### Bounded Queue Example (overwriteEnabled = FALSE)
```iecst
// Buffer capacity = 3
value := 100; ring.Push(value);  // Buffer: [100], returns TRUE
value := 200; ring.Push(value);  // Buffer: [100, 200], returns TRUE
value := 300; ring.Push(value);  // Buffer: [100, 200, 300], returns TRUE

// Push to full buffer fails
value := 400;
success := ring.Push(value);     // Returns FALSE, logs error, buffer unchanged
```

### Return Value
- **TRUE**: Element was successfully pushed to the ring buffer
- **FALSE**: Push operation failed (see error conditions)

### Error Conditions (both modes)
- Returns FALSE and logs error if buffer was not initialized
- Returns FALSE and logs error if element size doesn't match buffer element size
- Returns FALSE and logs error if underlying WriteAtIndex operation fails

### Error Conditions (overwriteEnabled = FALSE only)
- Returns FALSE and logs error if ring buffer is full (no available capacity)

### Parameters
- **element**: Must be a writable variable (not a literal) of the correct size
  - Must match the buffer's configured element size
  - Value will be copied into the ring buffer

### Side Effects (when not full)
- Adds one element to the ring buffer using WriteAtIndex
- Increments elementCount by 1 (managed by RingBuffer, not AnyBuffer)
- Advances tail pointer circularly
- Logs verbose trace message on success
- Logs error trace message on failure

### Side Effects (when full and overwriteEnabled = TRUE)
- Overwrites element at tail position using WriteAtIndex (no shifting!)
- Advances both head pointer and tail pointer circularly
- Element count remains at maximum capacity
- No physical element movement occurs
- No AnyBuffer counter modifications
- Logs verbose trace message on success

### Performance Considerations
- **When not full**: O(1) - uses WriteAtIndex (raw write, no counter overhead)
- **When full**: O(1) - uses WriteAtIndex with circular indexing (no shifting!)
- **Overall**: True O(1) constant-time operation for all scenarios
- **Optimal efficiency**: WriteAtIndex bypasses AnyBuffer counter management
- Ideal for high-frequency streaming and real-time data processing
*)
Push := FALSE;
IF NOT isInitialized THEN
	Trace.Error(__POUNAME(), 'Buffer was not initialized yet, execute method .init() at least once');
	RETURN;
END_IF

// valid sized element pushed?
IF element.diSize <> anyBuffer.Configuration.elementSize THEN
	Trace.Error(__POUNAME(), 'Pushed element is of improper size');
	RETURN;
END_IF

// Handle push based on buffer state
IF anyBuffer.Metadata.elementCount < anyBuffer.Configuration.capacity THEN
	// Buffer not yet full - use WriteAtIndex for direct write without counter changes
	Push := anyBuffer.ReplaceAtIndex(anyBuffer.Metadata.tailIndex, element);
	IF Push THEN
		// Advance tail circular
		AdvanceTail();

		// Replace index does not change counters, do it manually
		anyBuffer.Metadata.elementCount := anyBuffer.Metadata.elementCount + 1;
		anyBuffer.Metadata.capacity		:= anyBuffer.Metadata.capacity - 1;
	END_IF
ELSIF _overwrite THEN
	// Buffer is full and overwrite enabled - use WriteAtIndex for circular overwrite (no shifting!)
	Push := anyBuffer.ReplaceAtIndex(anyBuffer.Metadata.tailIndex, element);
	IF Push THEN
		// Advance tail circular
		AdvanceTail();

		// Advance head circular
		AdvanceHead();

		// elementCount stays at capacity
	END_IF
ELSE
	// Overwrite disabled - reject push when full (bounded queue behavior)
	Trace.Error(__POUNAME(), 'Attempt to push to full buffer with overwrite disabled');
	RETURN;
END_IF

// Push was ok, trace message
IF Push THEN
	Trace.Verbose(__POUNAME(), 'executed');
ELSE
	Trace.Error(__POUNAME(), 'FAILED');
END_IF
END_METHOD

END_FUNCTION_BLOCK

// Utilities/File/Interface/I_FileHandler
INTERFACE I_FileHandler EXTENDS I_Component, I_Cyclic, I_TaskResult, I_TaskResult, I_Resettable

METHOD ClearDocument
VAR_INPUT
END_VAR
END_METHOD

PROPERTY Datatype : T_MaxString
SET
END_SET
END_PROPERTY

METHOD LoadFile
END_METHOD

PROPERTY nData : UDINT
SET
END_SET
END_PROPERTY

PROPERTY PUBLIC Path : T_MaxString
GET
END_GET
SET
END_SET
END_PROPERTY

PROPERTY pData : PVOID
SET
END_SET
END_PROPERTY

METHOD ReadSymbol
END_METHOD

METHOD SaveFile
END_METHOD

PROPERTY SymbolName : T_MaxString
SET
END_SET
END_PROPERTY

PROPERTY Timeout : TIME
SET
END_SET
END_PROPERTY

METHOD UpdateSymbol
END_METHOD

END_INTERFACE

// Utilities/File/File_HMI
FUNCTION_BLOCK File_HMI EXTENDS HmiFunction
VAR
	File : I_FileHandler;
	{ attribute 'TcHmiSymbol.AddSymbol' }
	{ attribute 'TcHmiSymbol.AddSymbol.UserGroups' := '__SystemAdministrators,Admin' }
	File_HMI : ST_File_HMI;
END_VAR

PROPERTY LoadPermissive : I_Permissive
GET
LoadPermissive := File_HMI.Load.Permissive;
END_GET
END_PROPERTY

PROPERTY SavePermissive : I_Permissive
GET
SavePermissive := File_HMI.Save.Permissive;
END_GET
END_PROPERTY

PROPERTY ControlObject : I_Base
SET
__QueryInterface(ControlObject,File);
END_SET
END_PROPERTY

METHOD CyclicLogic
VAR_INST
	SaveRT		 : R_TRIG;
	LoadRT		 : R_TRIG;
	ReloadActive : BOOL;
END_VAR
IF File = 0 THEN
	RETURN;
END_IF

File_HMI.Name		:= File.Name;
File_HMI.HmiEnabled := Enabled;
// HMI Commands
IF Enabled THEN
	SaveRT(CLK := File_HMI.Save.Active);
	IF SaveRT.Q THEN
		IF File_HMI.Save.Permissive.OK THEN
			File.UpdateSymbol();
		END_IF
	END_IF

	IF ReloadActive AND NOT File.Busy AND NOT File.Error THEN
		File.ReadSymbol();
		ReloadActive := FALSE;
	END_IF

	LoadRT(CLK := File_HMI.Load.Active);
	IF LoadRT.Q THEN
		IF File_HMI.Load.Permissive.OK THEN
			File.LoadFile();
			ReloadActive := TRUE;
		END_IF
	END_IF

	IF File_HMI.NewPath THEN
		File.Path		 := File_HMI.Path;
		File_HMI.NewPath := FALSE;
	END_IF
END_IF
END_METHOD

(*FB_Init is always available implicitly and it is used primarily for initialization.
The return value is not evaluated. For a specific influence, you can also declare the
methods explicitly and provide additional code there with the standard initialization
code. You can evaluate the return value.*)
METHOD FB_Init : BOOL
VAR_INPUT
	(* TRUE: the retain variables are initialized (reset warm / reset cold)*)
	bInitRetains : BOOL;

	(* TRUE: the instance will be copied to the copy code afterward (online change)   *)
	bInCopyCode : BOOL;
	Name		: Core.T_MaxString;
	File		: I_FileHandler;
END_VAR
THIS^.File	:= File;
ControlType := 'File';
LinkObject	:= 'File_HMI';
END_METHOD

END_FUNCTION_BLOCK

// Utilities/File/JsonFile
FUNCTION_BLOCK JsonFile
VAR_GENERIC CONSTANT
	FileSize : UDINT := 10000;
END_VAR
EXTENDS CyclicComponent IMPLEMENTS I_FileHandler
VAR
	{attribute 'hide'}
	_Error : BOOL;
	{attribute 'hide'}
	_ErrorId : UDINT;

	//
	_Path	   : STRING;
	TonTimeout : TON;
	_Timeout   : TIME := T#1S;
	SeqLoad	   : UDINT;
	SeqSave	   : UDINT;

	// Folder Management
	CreateDir	 : FB_CreateDir;
	StringHelper : StringHelper;

	// Symbol
	JsonReadWriteDataType : FB_JsonReadWriteDatatype;
	ValueJson			  : STRING(FileSize);
	hr					  : HRESULT;
	_Datatype			  : T_MaxString;
	_SymbolName			  : T_MaxString;
	_nData				  : UDINT;
	_pData				  : PVOID;

	// Json Management 
	FileRead			  : BOOL;
	FileSave			  : BOOL;
	FileLoadOK			  : BOOL;
	FileSaveOK			  : BOOL;
	JsonFileMachineConfig : FB_JsonDomParser;
	JsonDoc				  : SJsonValue;
	JsonProp			  : SJsonValue;
END_VAR

METHOD CyclicLogic
IF _Path <> '' THEN
	FileLoadOK := JsonFileMachineConfig.LoadDocumentFromFile(sFile := _Path, bExec := FileRead);
	FileSaveOK := JsonFileMachineConfig.SaveDocumentToFile(sFile := _Path, bExec := FileSave);
END_IF

TonTimeout(IN := Busy, PT := _Timeout);
IF TonTimeout.Q THEN
	_Error := TRUE;
END_IF

SaveFileSequence();
LoadFileSequence();
END_METHOD

METHOD ClearDocument
VAR_INPUT
END_VAR
JsonDoc := JsonFileMachineConfig.NewDocument();
END_METHOD

PROPERTY Datatype : T_MaxString
SET
_Datatype := Datatype;
END_SET
END_PROPERTY

METHOD LoadFile
IF _Path = '' THEN
	_Error := TRUE;
	Trace.LogMessage(Name, 'File Path not set!');
	RETURN;
END_IF

IF Busy THEN
	RETURN;
END_IF

FileRead := TRUE;
SeqLoad	 := 10;
END_METHOD

PROPERTY nData : UDINT
SET
_nData := nData;
END_SET
END_PROPERTY

PROPERTY PUBLIC Path : T_MaxString
GET
Path := _Path;
END_GET
SET
//Prevent the path from have a space at the end
_Path := Path;
WHILE RIGHT(_Path, 1) = ' ' DO
	_Path := DELETE(_Path, 1, LEN(_Path));
END_WHILE
END_SET
END_PROPERTY

PROPERTY pData : PVOID
SET
_pData := pData;
END_SET
END_PROPERTY

METHOD ReadSymbol
IF JsonDoc = 0 THEN
	Trace.LogMessage(Name, 'Document File not loaded!');
	RETURN;
END_IF

IF _Datatype = '' THEN
	Trace.LogMessage(Name, 'No Datatype specified!');
	RETURN;
END_IF

IF _nData = 0 THEN
	Trace.LogMessage(Name, 'No nData specified!');
	RETURN;
END_IF

IF _pData = 0 THEN
	Trace.LogMessage(Name, 'No pData specified!');
	RETURN;
END_IF

IF _SymbolName = '' THEN
	Trace.LogMessage(Name, 'No PropertyName specified!');
	RETURN;
END_IF

IF Busy THEN
	RETURN;
END_IF

JsonProp := JsonFileMachineConfig.FindMemberPath(JsonDoc, _SymbolName);
JsonFileMachineConfig.CopyJson(v := JsonProp, pDoc := ValueJson, nDoc := SIZEOF(ValueJson));
IF JsonProp <> 0 THEN
	JsonReadWriteDataType.SetSymbolFromJson(sJson		:= ValueJson,
											sDataType	:= _Datatype,
											nData		:= _nData,
											pData		:= _pData,
											hrErrorCode => hr);
ELSE
	THIS^.UpdateSymbol();
END_IF
END_METHOD

METHOD SaveFile
IF _Path = '' THEN
	_Error := TRUE;
	Trace.LogMessage(Name, 'File Path not set!');
	RETURN;
END_IF

IF Busy THEN
	RETURN;
END_IF

FileSave := TRUE;
SeqSave	 := 10;
END_METHOD

PROPERTY SymbolName : T_MaxString
SET
_SymbolName := SymbolName;
END_SET
END_PROPERTY

PROPERTY Timeout : TIME
SET
_Timeout := Timeout;
END_SET
END_PROPERTY

METHOD UpdateSymbol
IF JsonDoc = 0 THEN
	Trace.LogMessage(Name, 'Document File not loaded!');
	RETURN;
END_IF

IF _Datatype = '' THEN
	Trace.LogMessage(Name, 'No Datatype specified!');
	RETURN;
END_IF

IF _nData = 0 THEN
	Trace.LogMessage(Name, 'No nData specified!');
	RETURN;
END_IF

IF _pData = 0 THEN
	Trace.LogMessage(Name, 'No pData specified!');
	RETURN;
END_IF

IF _SymbolName = '' THEN
	Trace.LogMessage(Name, 'No PropertyName specified!');
	RETURN;
END_IF

IF Busy THEN
	RETURN;
END_IF

// Create Json
JsonReadWriteDataType.CopyJsonStringFromSymbol(sDatatype   := _Datatype,
											   nData	   := _nData,
											   pData	   := _pData,
											   pDoc		   := ValueJson,
											   nDoc		   := SIZEOF(ValueJson),
											   hrErrorCode => hr);

// Attempt to find Member
jsonProp := JsonFileMachineConfig.FindMemberPath(JsonDoc, _SymbolName);
IF JsonProp <> 0 THEN
	JsonFileMachineConfig.SetJson(JsonProp, ValueJson);
ELSE
	JsonFileMachineConfig.AddJsonMember(JsonDoc, _SymbolName, ValueJson);
END_IF

// Save the update to file
FileSave := TRUE;
SeqSave	 := 10;
JsonProp := 0;
END_METHOD

METHOD PRIVATE LoadFileSequence
VAR_INST
	dirPath	 : T_MaxString;
	tryAgain : BOOL;
END_VAR

VAR
	msg : STRING;
END_VAR
CASE SeqLoad OF
	0:										// Attempt to Load File -> Command started in LoadFile()
	10:										// Load File Done
		IF NOT FileRead AND FileLoadOK THEN // File Found
			JsonDoc := JsonFileMachineConfig.GetDocumentRoot();
			SeqLoad := 0;
		END_IF

		IF (NOT FileRead AND NOT FileLoadOK) OR TonTimeout.Q THEN // File not Found
			tryAgain := FALSE;
			FileRead := FALSE;
			SeqLoad	 := 20;
		END_IF

	20:								  (*File Not Found - Create Directory if not exists*) ;
		CreateDir(bExecute := FALSE); //Prepare for rising edge in next step
		IF NOT tryAgain THEN
			dirPath := StringHelper.GetPath(_Path);
		ELSE
			dirPath := StringHelper.GetPath(dirPath);
		END_IF

		SeqLoad := 30;

	30:
		CreateDir(sNetId	:= '',
				  sPathName := dirPath,
				  ePath		:= PATH_GENERIC,
				  bExecute	:= TRUE);

		IF NOT CreateDir.bBusy THEN
			IF NOT CreateDir.bError THEN
				IF NOT tryAgain THEN
					SeqLoad := 40;
				ELSE
					tryAgain := FALSE;
					SeqLoad	 := 20;
				END_IF
			ELSE
				IF (CreateDir.nErrId = 1827) OR (CreateDir.nErrId = 1807) THEN
					//0x723 Folder is already existing or invalid sPathName or ePath parameter.
					msg := CONCAT(_Path, ' File not found, but folder is existing. File will be created');
					Trace.LogMessage(Name, msg);
					SeqLoad := 40;
				ELSIF CreateDir.nErrId = 1804 THEN
					//0x70C Folder not found.
					msg := CONCAT('Folder is not found: ', dirPath);
					msg := CONCAT(msg, ' Reducing Path and trying again.');
					Trace.LogMessage(Name, msg);
					tryagain := TRUE;

					// SeqLoad	 := 20; TwinCat Bug - Ticket BTS-168764 Germany
					SeqLoad := 40;
				ELSE
					msg := CONCAT('Create Directory Error: ', UDINT_TO_STRING(CreateDir.nErrId));
					Trace.LogMessage(Name, msg);
					SeqLoad := 999;
				END_IF
			END_IF
		END_IF

	40: // File not found -> Create file
		JsonDoc	 := JsonFileMachineConfig.NewDocument();
		FileSave := TRUE;
		SeqLoad	 := 50;

	50: // New Document Saved
		IF NOT FileSave AND FileSaveOk THEN
			_Error	:= FALSE;
			SeqLoad := 0;
		END_IF
END_CASE
END_METHOD

METHOD PRIVATE SaveFileSequence
CASE SeqSave OF
	0:	// Attempt to save File -> Command started in UpdateXYZ()
	10: // New Document Saved
		IF NOT FileSave AND FileSaveOk THEN
			SeqSave := 0;
		END_IF
END_CASE
END_METHOD

METHOD Reset
_Error		  := FALSE;
_ErrorId	  := 0;
SeqSave		  := 0;
SeqLoad		  := 0;
TonTimeout.IN := FALSE;
END_METHOD

{attribute 'monitoring' := 'call'}
PROPERTY Busy : BOOL
GET
Busy := SeqSave <> 0 OR SeqLoad <> 0;
END_GET
END_PROPERTY

{attribute 'monitoring' := 'call'}
PROPERTY Error : BOOL
GET
Error := _Error;
END_GET
END_PROPERTY

{attribute 'monitoring' := 'call'}
PROPERTY ErrorId : UDINT
GET
ErrorID := _ErrorID;
END_GET
END_PROPERTY

END_FUNCTION_BLOCK

// Utilities/File/StringHelper
{attribute 'no_explicit_call' := 'This FB is a CLASS and must be accessed using methods or properties'}
FUNCTION_BLOCK StringHelper

METHOD PROTECTED GetExtensionOrVarName : T_MaxString
VAR_INPUT
	input : T_MaxString;
END_VAR

VAR
	i		 : INT;
	charArry : ARRAY[0..255] OF STRING(1);
END_VAR
IF NOT ValidInput(input) THEN
	RETURN;
END_IF

charArry := StringToCharArray(input);
//Get Location of final delimiter '.'
FOR i := LEN(input) - 1 TO 0 BY -1 DO //Start at the end and find the last delimiter
	IF charArry[i] = '.' THEN
		GetExtensionOrVarName := RIGHT(input, LEN(input) - 1 - i);
		EXIT;
	END_IF
END_FOR
END_METHOD

METHOD PROTECTED GetFileNameFromPath : T_MaxString
VAR_INPUT
	input : T_MaxString;
END_VAR

VAR
	i			  : INT;
	searchResults : ARRAY[0..99] OF INT;
	tempPath	  : T_MaxString;
END_VAR
IF NOT ValidInput(input) THEN
	RETURN;
END_IF

tempPath := input; //Copy to temp variable for modification
FOR i := 0 TO LEN(input) - 1 DO
	searchResults[i] := FIND(tempPath, '\');
	IF searchResults[i] > 0 THEN
		tempPath := RIGHT(tempPath, LEN(tempPath) - searchResults[i]); //Remove begining up to and including the first delimiter
	ELSE
		EXIT; //No more delimiters remaining
	END_IF
END_FOR

GetFileNameFromPath := tempPath;
END_METHOD

METHOD PROTECTED GetFilePath : T_MaxString
VAR_INPUT
	input : T_MaxString;
END_VAR

VAR
	tempPath	  : T_MaxString;
	i			  : INT;
	searchResults : ARRAY[0..99] OF INT;
	location	  : INT;
END_VAR
IF NOT ValidInput(input) THEN
	RETURN;
END_IF

tempPath := input;								 //Copy to temp variable for modification
tempPath := LEFT(tempPath, (LEN(tempPath) - 1)); //Remove Last Character, on first pass this has no effect, but on subsequents passes this will remove the ending \

//Reduce String by removing each delimiter and counting number of characters removed to find last '\'
FOR i := 0 TO LEN(input) - 1 DO
	searchResults[i] := FIND(tempPath, '\');
	IF searchResults[i] > 0 THEN
		tempPath := RIGHT(tempPath, LEN(tempPath) - searchResults[i]); //Remove begining up to and including the first delimiter
	ELSE
		EXIT; //No more delimiters remaining
	END_IF
END_FOR

//Sum length of string to last delimiter
FOR i := 0 TO LEN(input) - 1 DO
	IF searchResults[i] > 0 THEN
		location := location + searchResults[i]; //Location of last delimiter
	ELSE
		EXIT;
	END_IF
END_FOR

GetFilePath := LEFT(input, location);
END_METHOD

METHOD GetName : T_MaxString
VAR_INPUT
	FullPath : T_MaxString;
END_VAR
IF NOT ValidInput(FullPath) THEN
	RETURN;
END_IF

//Find the First \ or . to determine if this is a File Path or Symbol Path
IF FIND(FullPath, '\') > 0 THEN
	GetName := GetFileNameFromPath(FullPath);
ELSE //symbolPath
	GetName := GetExtensionOrVarName(FullPath);
END_IF
END_METHOD

METHOD GetPath : T_MaxString
VAR_INPUT
	FullPath : T_MaxString;
END_VAR

VAR
	tempPath : T_MaxString;
END_VAR
IF NOT ValidInput(FullPath) THEN
	RETURN;
END_IF

//Find the First \ or . to determine if this is a File Path or Symbol Path
IF FIND(FullPath, '\') > 0 THEN
	GetPath := GetFilePath(FullPath);
ELSE //symbolPath
	GetPath := GetSymbolPath(FullPath);
END_IF
END_METHOD

METHOD PROTECTED GetSymbolPath : T_MaxString
VAR_INPUT
	input : T_MaxString;
END_VAR

VAR
	i		 : INT;
	charArry : ARRAY[0..255] OF STRING(1);
	tempPath : T_MaxString;
END_VAR
IF NOT ValidInput(input) THEN
	RETURN;
END_IF

charArry := StringToCharArray(input);
tempPath := input;					  //Copy to temp variable for modification
FOR i := LEN(input) - 1 TO 0 BY -1 DO //Start at the end and find the last delimiter
	IF charArry[i] = '.' THEN
		tempPath := LEFT(tempPath, i);
		EXIT;
	END_IF
END_FOR

GetSymbolPath := tempPath;
END_METHOD

METHOD PROTECTED RemoveFirstChar : T_MaxString
VAR_INPUT
	input : T_MaxString;
END_VAR
RemoveFirstChar := DELETE(input, 1, 1);
END_METHOD

METHOD PROTECTED RemoveLastChar : T_MaxString
VAR_INPUT
	input : T_MaxString;
END_VAR
RemoveLastChar := DELETE(input, 1, len(input));
END_METHOD

METHOD PROTECTED StringToCharArray : ARRAY[0..255] OF STRING(1)
VAR_INPUT
	input : T_MaxString;
END_VAR

VAR
	i		 : INT;
	end		 : INT;
	tempPath : T_MaxString;
END_VAR
IF NOT ValidInput(input) THEN
	RETURN;
END_IF

tempPath := input;
//Convert String to CharArray
FOR i := 0 TO LEN(input) - 1 DO
	StringToCharArray[i] := Left(tempPath, 1); //Return the first/next character
	tempPath			 := RemoveFirstChar(tempPath);
END_FOR
END_METHOD

METHOD PROTECTED ValidInput : BOOL
VAR_INPUT
	input : T_MaxString;
END_VAR
IF LEN(input) > 0 THEN
	ValidInput := TRUE;
ELSE
	ValidInput := FALSE;
END_IF
END_METHOD

END_FUNCTION_BLOCK

// Utilities/Flash/SyncedSquareWaves
FUNCTION_BLOCK SyncedSquareWaves EXTENDS CyclicComponent IMPLEMENTS I_Initializable
VAR
	_Initialized  : BOOL;
	PLC_CycleTime : UDINT;
	CycleTime_ms  : LREAL;

	//
	{attribute 'hide'}
	_Wave_500Hz : BOOL;
	{attribute 'hide'}
	_Wave_100Hz : BOOL;
	{attribute 'hide'}
	_Wave_50Hz : BOOL;
	{attribute 'hide'}
	_Wave_5Hz : BOOL;
	{attribute 'hide'}
	_Wave_2Hz : BOOL;
	{attribute 'hide'}
	_Wave_1Hz : BOOL;
	{attribute 'hide'}
	_Wave_0_5Hz : BOOL;
END_VAR

METHOD Initialize
//PLC Scan Info
PLC_CycleTime := TwinCAT_SystemInfoVarList._TaskInfo[GETCURTASKINDEXEX()].CycleTime;
CycleTime_ms  := TO_LREAL(PLC_CycleTime) / 10000.0;

//
_Wave_500Hz	 := TRUE;
_Wave_100Hz	 := TRUE;
_Wave_50Hz	 := TRUE;
_Wave_5Hz	 := TRUE;
_Wave_2Hz	 := TRUE;
_Wave_1Hz	 := TRUE;
_Wave_0_5Hz	 := TRUE;
_Initialized := TRUE;
END_METHOD

{attribute 'monitoring' := 'call'}
PROPERTY Initialized : BOOL
GET
Initialized := _Initialized;
END_GET
SET
_Initialized := Initialized;
END_SET
END_PROPERTY

//! @summary This method serves as the entry point for all underlying FB logic
METHOD PUBLIC CyclicLogic
VAR
	Counter		   : LREAL;
	CountsRequired : LREAL;
	CycleCount	   : UDINT;
END_VAR
IF NOT _Initialized THEN
	Initialize();
	RETURN;
END_IF

CycleCount := TwinCAT_SystemInfoVarList._TaskInfo[GETCURTASKINDEXEX()].CycleCount;
IF (CycleTime_ms <= 1) AND (FRAC(1 / CycleTime_ms) = 0) THEN
	CountsRequired := 1 / CycleTime_ms;
	Counter		   := LMOD(CycleCount, CountsRequired);
	IF (Counter + 1) = CountsRequired THEN
		_Wave_500Hz := NOT _Wave_500Hz;
	END_IF
END_IF

IF (CycleTime_ms <= 5) AND (FRAC(5 / CycleTime_ms) = 0) THEN
	CountsRequired := 5 / CycleTime_ms;
	Counter		   := LMOD(CycleCount, CountsRequired);
	IF (Counter + 1) = CountsRequired THEN
		_Wave_100Hz := NOT _Wave_100Hz;
	END_IF
END_IF

IF (CycleTime_ms <= 10) AND (FRAC(10 / CycleTime_ms) = 0) THEN
	CountsRequired := 10 / CycleTime_ms;
	Counter		   := LMOD(CycleCount, CountsRequired);
	IF (Counter + 1) = CountsRequired THEN
		_Wave_50Hz := NOT _Wave_50Hz;
	END_IF
END_IF

IF (CycleTime_ms <= 100) AND (FRAC(100 / CycleTime_ms) = 0) THEN
	CountsRequired := 100 / CycleTime_ms;
	Counter		   := LMOD(CycleCount, CountsRequired);
	IF (Counter + 1) = CountsRequired THEN
		_Wave_5Hz := NOT _Wave_5Hz;
	END_IF
END_IF

IF (CycleTime_ms <= 250) AND (FRAC(250 / CycleTime_ms) = 0) THEN
	CountsRequired := 250 / CycleTime_ms;
	Counter		   := LMOD(CycleCount, CountsRequired);
	IF (Counter + 1) = CountsRequired THEN
		_Wave_2Hz := NOT _Wave_2Hz;
	END_IF
END_IF

IF (CycleTime_ms <= 500) AND (FRAC(500 / CycleTime_ms) = 0) THEN
	CountsRequired := 500 / CycleTime_ms;
	Counter		   := LMOD(CycleCount, CountsRequired);
	IF (Counter + 1) = CountsRequired THEN
		_Wave_1Hz := NOT _Wave_1Hz;
	END_IF
END_IF

IF (CycleTime_ms <= 1000) AND (FRAC(1000 / CycleTime_ms) = 0) THEN
	CountsRequired := 1000 / CycleTime_ms;
	Counter		   := LMOD(CycleCount, CountsRequired);
	IF (Counter + 1) = CountsRequired THEN
		_Wave_0_5Hz := NOT _Wave_0_5Hz;
	END_IF
END_IF
END_METHOD

{attribute 'monitoring' := 'call'}
PROPERTY Wave_0_5Hz : BOOL
GET
Wave_0_5Hz := _Wave_0_5Hz;
END_GET
END_PROPERTY

{attribute 'monitoring' := 'call'}
PROPERTY Wave_100Hz : BOOL
GET
Wave_100Hz := _Wave_100Hz;
END_GET
END_PROPERTY

{attribute 'monitoring' := 'call'}
PROPERTY Wave_1Hz : BOOL
GET
Wave_1Hz := _Wave_1Hz;
END_GET
END_PROPERTY

{attribute 'monitoring' := 'call'}
PROPERTY Wave_2Hz : BOOL
GET
Wave_2Hz := _Wave_2Hz;
END_GET
END_PROPERTY

{attribute 'monitoring' := 'call'}
PROPERTY Wave_500Hz : BOOL
GET
Wave_500Hz := _Wave_500Hz;
END_GET
END_PROPERTY

{attribute 'monitoring' := 'call'}
PROPERTY Wave_50Hz : BOOL
GET
Wave_50Hz := _Wave_50Hz;
END_GET
END_PROPERTY

{attribute 'monitoring' := 'call'}
PROPERTY Wave_5Hz : BOOL
GET
Wave_5Hz := _Wave_5Hz;
END_GET
END_PROPERTY

END_FUNCTION_BLOCK

// Utilities/Functions/CompareLREAL
FUNCTION CompareLREAL : BOOL
VAR_INPUT
	Var1	: LREAL;
	Var2	: LREAL;
	Epsilon : LREAL := 1E-6;
END_VAR

CompareLREAL := ABS(Var1 - Var2) < Epsilon;

END_FUNCTION

// Utilities/Functions/CompareModulo
FUNCTION CompareModulo : BOOL
VAR_INPUT
	Var1	: LREAL;
	Var2	: LREAL;
	Modulo	: LREAL := 360.0;
	Epsilon : LREAL := 1E-6;
END_VAR

CompareModulo := (ABS(MODABS(Var1, Modulo) - MODABS(Var2, Modulo)) < Epsilon) OR (ABS(MODABS(Var1, Modulo) - MODABS(Var2, Modulo)) > (Modulo - Epsilon));

END_FUNCTION

// Utilities/Functions/PercentToAnalog
FUNCTION PercentToAnalog : INT
VAR_INPUT
	TargetValue : DINT; // 0-100%
END_VAR

PercentToAnalog := TO_INT(32767 * TargetValue / 100);

END_FUNCTION

// Utilities/Timing/Stopwatch
FUNCTION_BLOCK Stopwatch
VAR
	StartTime			: T_DCTIME64;
	EndTime				: T_DCTIME64;
	PreviousLapEndTime	: T_DCTIME64;
	PreviousElapsedTime : LREAL;
	_Running			: BOOL;
END_VAR

VAR CONSTANT
	OneNanosecond : LREAL := 1.0E-9;
END_VAR

{attribute 'monitoring' := 'call'}
PROPERTY Elapsed : LREAL
GET
IF _Running THEN
	Elapsed := TO_LREAL(F_GetCurDcTickTime64() - StartTime) * OneNanosecond;
ELSE
	Elapsed := PreviousElapsedTime;
END_IF
END_GET
END_PROPERTY

METHOD Lap : LREAL;
VAR
	LapEndTime	: T_DCTIME64;
	LapDuration : LREAL;
END_VAR
IF _Running THEN
	LapEndTime		   := F_GetActualDcTime64();
	LapDuration		   := TO_LREAL(LapEndTime - PreviousLapEndTime) * OneNanosecond;
	PreviousLapEndTime := LapEndTime;
	Lap				   := LapDuration;
END_IF
END_METHOD

{attribute 'monitoring' := 'call'}
PROPERTY Running : BOOL
GET
Running := _Running;
END_GET
END_PROPERTY

METHOD Start
StartTime			:= F_GetActualDcTime64();
PreviousLapEndTime	:= StartTime;
_Running			:= TRUE;
PreviousElapsedTime := 0.0;
PreviousElapsedTime := 0;
END_METHOD

METHOD Stop : LREAL
IF _Running THEN
	EndTime				:= F_GetActualDcTime64();
	_Running			:= FALSE;
	PreviousElapsedTime := TO_LREAL(EndTime - StartTime) * OneNanosecond;
	Stop				:= PreviousElapsedTime;
ELSE
	Stop := 0.0;
END_IF
END_METHOD

END_FUNCTION_BLOCK
